FUNCTION_BLOCK ASSEMBLE_AL_FROM_AX (* this Function combines the 64 AX (BOOL) adapters to a AL (LWORD) *)
  (* Standard: 61499-2; Description: Copyright (c) 2026 Meisterschulen am Ostbahnhof SPDX-License-Identifier: EPL-2.0 *)
  (* Version 1.0, 2026-05-16, Franz Höpfinger, Meisterschulen am Ostbahnhof, initial API and implementation and/or initial documentation *)
  PACKAGE adapter::assembling;
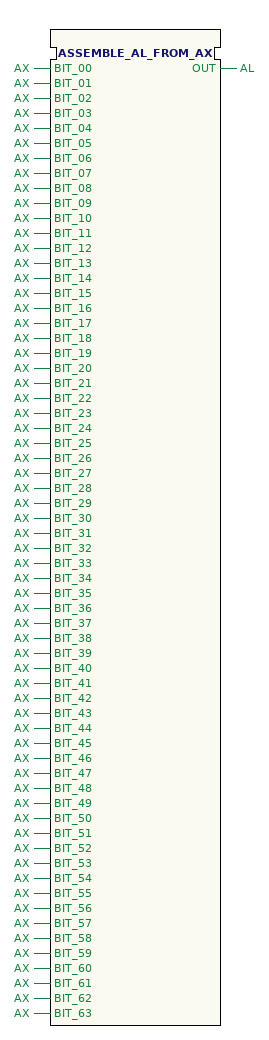
  SOCKETS
    BIT_00 : adapter::types::unidirectional::AX; (* Bool Bit 0 *)
    BIT_01 : adapter::types::unidirectional::AX; (* Bool Bit 1 *)
    BIT_02 : adapter::types::unidirectional::AX; (* Bool Bit 2 *)
    BIT_03 : adapter::types::unidirectional::AX; (* Bool Bit 3 *)
    BIT_04 : adapter::types::unidirectional::AX; (* Bool Bit 4 *)
    BIT_05 : adapter::types::unidirectional::AX; (* Bool Bit 5 *)
    BIT_06 : adapter::types::unidirectional::AX; (* Bool Bit 6 *)
    BIT_07 : adapter::types::unidirectional::AX; (* Bool Bit 7 *)
    BIT_08 : adapter::types::unidirectional::AX; (* Bool Bit 8 *)
    BIT_09 : adapter::types::unidirectional::AX; (* Bool Bit 9 *)
    BIT_10 : adapter::types::unidirectional::AX; (* Bool Bit 10 *)
    BIT_11 : adapter::types::unidirectional::AX; (* Bool Bit 11 *)
    BIT_12 : adapter::types::unidirectional::AX; (* Bool Bit 12 *)
    BIT_13 : adapter::types::unidirectional::AX; (* Bool Bit 13 *)
    BIT_14 : adapter::types::unidirectional::AX; (* Bool Bit 14 *)
    BIT_15 : adapter::types::unidirectional::AX; (* Bool Bit 15 *)
    BIT_16 : adapter::types::unidirectional::AX; (* Bool Bit 16 *)
    BIT_17 : adapter::types::unidirectional::AX; (* Bool Bit 17 *)
    BIT_18 : adapter::types::unidirectional::AX; (* Bool Bit 18 *)
    BIT_19 : adapter::types::unidirectional::AX; (* Bool Bit 19 *)
    BIT_20 : adapter::types::unidirectional::AX; (* Bool Bit 20 *)
    BIT_21 : adapter::types::unidirectional::AX; (* Bool Bit 21 *)
    BIT_22 : adapter::types::unidirectional::AX; (* Bool Bit 22 *)
    BIT_23 : adapter::types::unidirectional::AX; (* Bool Bit 23 *)
    BIT_24 : adapter::types::unidirectional::AX; (* Bool Bit 24 *)
    BIT_25 : adapter::types::unidirectional::AX; (* Bool Bit 25 *)
    BIT_26 : adapter::types::unidirectional::AX; (* Bool Bit 26 *)
    BIT_27 : adapter::types::unidirectional::AX; (* Bool Bit 27 *)
    BIT_28 : adapter::types::unidirectional::AX; (* Bool Bit 28 *)
    BIT_29 : adapter::types::unidirectional::AX; (* Bool Bit 29 *)
    BIT_30 : adapter::types::unidirectional::AX; (* Bool Bit 30 *)
    BIT_31 : adapter::types::unidirectional::AX; (* Bool Bit 31 *)
    BIT_32 : adapter::types::unidirectional::AX; (* Bool Bit 32 *)
    BIT_33 : adapter::types::unidirectional::AX; (* Bool Bit 33 *)
    BIT_34 : adapter::types::unidirectional::AX; (* Bool Bit 34 *)
    BIT_35 : adapter::types::unidirectional::AX; (* Bool Bit 35 *)
    BIT_36 : adapter::types::unidirectional::AX; (* Bool Bit 36 *)
    BIT_37 : adapter::types::unidirectional::AX; (* Bool Bit 37 *)
    BIT_38 : adapter::types::unidirectional::AX; (* Bool Bit 38 *)
    BIT_39 : adapter::types::unidirectional::AX; (* Bool Bit 39 *)
    BIT_40 : adapter::types::unidirectional::AX; (* Bool Bit 40 *)
    BIT_41 : adapter::types::unidirectional::AX; (* Bool Bit 41 *)
    BIT_42 : adapter::types::unidirectional::AX; (* Bool Bit 42 *)
    BIT_43 : adapter::types::unidirectional::AX; (* Bool Bit 43 *)
    BIT_44 : adapter::types::unidirectional::AX; (* Bool Bit 44 *)
    BIT_45 : adapter::types::unidirectional::AX; (* Bool Bit 45 *)
    BIT_46 : adapter::types::unidirectional::AX; (* Bool Bit 46 *)
    BIT_47 : adapter::types::unidirectional::AX; (* Bool Bit 47 *)
    BIT_48 : adapter::types::unidirectional::AX; (* Bool Bit 48 *)
    BIT_49 : adapter::types::unidirectional::AX; (* Bool Bit 49 *)
    BIT_50 : adapter::types::unidirectional::AX; (* Bool Bit 50 *)
    BIT_51 : adapter::types::unidirectional::AX; (* Bool Bit 51 *)
    BIT_52 : adapter::types::unidirectional::AX; (* Bool Bit 52 *)
    BIT_53 : adapter::types::unidirectional::AX; (* Bool Bit 53 *)
    BIT_54 : adapter::types::unidirectional::AX; (* Bool Bit 54 *)
    BIT_55 : adapter::types::unidirectional::AX; (* Bool Bit 55 *)
    BIT_56 : adapter::types::unidirectional::AX; (* Bool Bit 56 *)
    BIT_57 : adapter::types::unidirectional::AX; (* Bool Bit 57 *)
    BIT_58 : adapter::types::unidirectional::AX; (* Bool Bit 58 *)
    BIT_59 : adapter::types::unidirectional::AX; (* Bool Bit 59 *)
    BIT_60 : adapter::types::unidirectional::AX; (* Bool Bit 60 *)
    BIT_61 : adapter::types::unidirectional::AX; (* Bool Bit 61 *)
    BIT_62 : adapter::types::unidirectional::AX; (* Bool Bit 62 *)
    BIT_63 : adapter::types::unidirectional::AX; (* Bool Bit 63 *)
  END_SOCKETS
  PLUGS
    OUT : adapter::types::unidirectional::AL; (* LWORD Output *)
  END_PLUGS
  FBS
    ASSEMBLE_LWORD_FROM_BOOLS : eclipse4diac::utils::assembling::ASSEMBLE_LWORD_FROM_BOOLS;
    E_D_FF_ANY : iec61499::events::E_D_FF_ANY;
  END_FBS
  EVENT_CONNECTIONS
    BIT_00.E1 TO ASSEMBLE_LWORD_FROM_BOOLS.REQ;
    BIT_01.E1 TO ASSEMBLE_LWORD_FROM_BOOLS.REQ;
    BIT_02.E1 TO ASSEMBLE_LWORD_FROM_BOOLS.REQ;
    BIT_03.E1 TO ASSEMBLE_LWORD_FROM_BOOLS.REQ;
    BIT_04.E1 TO ASSEMBLE_LWORD_FROM_BOOLS.REQ;
    BIT_05.E1 TO ASSEMBLE_LWORD_FROM_BOOLS.REQ;
    BIT_06.E1 TO ASSEMBLE_LWORD_FROM_BOOLS.REQ;
    BIT_07.E1 TO ASSEMBLE_LWORD_FROM_BOOLS.REQ;
    BIT_08.E1 TO ASSEMBLE_LWORD_FROM_BOOLS.REQ;
    BIT_09.E1 TO ASSEMBLE_LWORD_FROM_BOOLS.REQ;
    BIT_10.E1 TO ASSEMBLE_LWORD_FROM_BOOLS.REQ;
    BIT_11.E1 TO ASSEMBLE_LWORD_FROM_BOOLS.REQ;
    BIT_12.E1 TO ASSEMBLE_LWORD_FROM_BOOLS.REQ;
    BIT_13.E1 TO ASSEMBLE_LWORD_FROM_BOOLS.REQ;
    BIT_14.E1 TO ASSEMBLE_LWORD_FROM_BOOLS.REQ;
    BIT_15.E1 TO ASSEMBLE_LWORD_FROM_BOOLS.REQ;
    BIT_16.E1 TO ASSEMBLE_LWORD_FROM_BOOLS.REQ;
    BIT_17.E1 TO ASSEMBLE_LWORD_FROM_BOOLS.REQ;
    BIT_18.E1 TO ASSEMBLE_LWORD_FROM_BOOLS.REQ;
    BIT_19.E1 TO ASSEMBLE_LWORD_FROM_BOOLS.REQ;
    BIT_20.E1 TO ASSEMBLE_LWORD_FROM_BOOLS.REQ;
    BIT_21.E1 TO ASSEMBLE_LWORD_FROM_BOOLS.REQ;
    BIT_22.E1 TO ASSEMBLE_LWORD_FROM_BOOLS.REQ;
    BIT_23.E1 TO ASSEMBLE_LWORD_FROM_BOOLS.REQ;
    BIT_24.E1 TO ASSEMBLE_LWORD_FROM_BOOLS.REQ;
    BIT_25.E1 TO ASSEMBLE_LWORD_FROM_BOOLS.REQ;
    BIT_26.E1 TO ASSEMBLE_LWORD_FROM_BOOLS.REQ;
    BIT_27.E1 TO ASSEMBLE_LWORD_FROM_BOOLS.REQ;
    BIT_28.E1 TO ASSEMBLE_LWORD_FROM_BOOLS.REQ;
    BIT_29.E1 TO ASSEMBLE_LWORD_FROM_BOOLS.REQ;
    BIT_30.E1 TO ASSEMBLE_LWORD_FROM_BOOLS.REQ;
    BIT_31.E1 TO ASSEMBLE_LWORD_FROM_BOOLS.REQ;
    BIT_32.E1 TO ASSEMBLE_LWORD_FROM_BOOLS.REQ;
    BIT_33.E1 TO ASSEMBLE_LWORD_FROM_BOOLS.REQ;
    BIT_34.E1 TO ASSEMBLE_LWORD_FROM_BOOLS.REQ;
    BIT_35.E1 TO ASSEMBLE_LWORD_FROM_BOOLS.REQ;
    BIT_36.E1 TO ASSEMBLE_LWORD_FROM_BOOLS.REQ;
    BIT_37.E1 TO ASSEMBLE_LWORD_FROM_BOOLS.REQ;
    BIT_38.E1 TO ASSEMBLE_LWORD_FROM_BOOLS.REQ;
    BIT_39.E1 TO ASSEMBLE_LWORD_FROM_BOOLS.REQ;
    BIT_40.E1 TO ASSEMBLE_LWORD_FROM_BOOLS.REQ;
    BIT_41.E1 TO ASSEMBLE_LWORD_FROM_BOOLS.REQ;
    BIT_42.E1 TO ASSEMBLE_LWORD_FROM_BOOLS.REQ;
    BIT_43.E1 TO ASSEMBLE_LWORD_FROM_BOOLS.REQ;
    BIT_44.E1 TO ASSEMBLE_LWORD_FROM_BOOLS.REQ;
    BIT_45.E1 TO ASSEMBLE_LWORD_FROM_BOOLS.REQ;
    BIT_46.E1 TO ASSEMBLE_LWORD_FROM_BOOLS.REQ;
    BIT_47.E1 TO ASSEMBLE_LWORD_FROM_BOOLS.REQ;
    BIT_48.E1 TO ASSEMBLE_LWORD_FROM_BOOLS.REQ;
    BIT_49.E1 TO ASSEMBLE_LWORD_FROM_BOOLS.REQ;
    BIT_50.E1 TO ASSEMBLE_LWORD_FROM_BOOLS.REQ;
    BIT_51.E1 TO ASSEMBLE_LWORD_FROM_BOOLS.REQ;
    BIT_52.E1 TO ASSEMBLE_LWORD_FROM_BOOLS.REQ;
    BIT_53.E1 TO ASSEMBLE_LWORD_FROM_BOOLS.REQ;
    BIT_54.E1 TO ASSEMBLE_LWORD_FROM_BOOLS.REQ;
    BIT_55.E1 TO ASSEMBLE_LWORD_FROM_BOOLS.REQ;
    BIT_56.E1 TO ASSEMBLE_LWORD_FROM_BOOLS.REQ;
    BIT_57.E1 TO ASSEMBLE_LWORD_FROM_BOOLS.REQ;
    BIT_58.E1 TO ASSEMBLE_LWORD_FROM_BOOLS.REQ;
    BIT_59.E1 TO ASSEMBLE_LWORD_FROM_BOOLS.REQ;
    BIT_60.E1 TO ASSEMBLE_LWORD_FROM_BOOLS.REQ;
    BIT_61.E1 TO ASSEMBLE_LWORD_FROM_BOOLS.REQ;
    BIT_62.E1 TO ASSEMBLE_LWORD_FROM_BOOLS.REQ;
    BIT_63.E1 TO ASSEMBLE_LWORD_FROM_BOOLS.REQ;
    ASSEMBLE_LWORD_FROM_BOOLS.CNF TO E_D_FF_ANY.CLK;
    E_D_FF_ANY.EO TO OUT.E1;
  END_CONNECTIONS
  DATA_CONNECTIONS
    ASSEMBLE_LWORD_FROM_BOOLS. TO E_D_FF_ANY.D;
    E_D_FF_ANY.Q TO OUT.D1;
    BIT_63.D1 TO ASSEMBLE_LWORD_FROM_BOOLS.BIT_63;
    BIT_62.D1 TO ASSEMBLE_LWORD_FROM_BOOLS.BIT_62;
    BIT_61.D1 TO ASSEMBLE_LWORD_FROM_BOOLS.BIT_61;
    BIT_60.D1 TO ASSEMBLE_LWORD_FROM_BOOLS.BIT_60;
    BIT_59.D1 TO ASSEMBLE_LWORD_FROM_BOOLS.BIT_59;
    BIT_58.D1 TO ASSEMBLE_LWORD_FROM_BOOLS.BIT_58;
    BIT_57.D1 TO ASSEMBLE_LWORD_FROM_BOOLS.BIT_57;
    BIT_56.D1 TO ASSEMBLE_LWORD_FROM_BOOLS.BIT_56;
    BIT_55.D1 TO ASSEMBLE_LWORD_FROM_BOOLS.BIT_55;
    BIT_54.D1 TO ASSEMBLE_LWORD_FROM_BOOLS.BIT_54;
    BIT_53.D1 TO ASSEMBLE_LWORD_FROM_BOOLS.BIT_53;
    BIT_52.D1 TO ASSEMBLE_LWORD_FROM_BOOLS.BIT_52;
    BIT_51.D1 TO ASSEMBLE_LWORD_FROM_BOOLS.BIT_51;
    BIT_50.D1 TO ASSEMBLE_LWORD_FROM_BOOLS.BIT_50;
    BIT_49.D1 TO ASSEMBLE_LWORD_FROM_BOOLS.BIT_49;
    BIT_48.D1 TO ASSEMBLE_LWORD_FROM_BOOLS.BIT_48;
    BIT_47.D1 TO ASSEMBLE_LWORD_FROM_BOOLS.BIT_47;
    BIT_46.D1 TO ASSEMBLE_LWORD_FROM_BOOLS.BIT_46;
    BIT_45.D1 TO ASSEMBLE_LWORD_FROM_BOOLS.BIT_45;
    BIT_44.D1 TO ASSEMBLE_LWORD_FROM_BOOLS.BIT_44;
    BIT_43.D1 TO ASSEMBLE_LWORD_FROM_BOOLS.BIT_43;
    BIT_42.D1 TO ASSEMBLE_LWORD_FROM_BOOLS.BIT_42;
    BIT_41.D1 TO ASSEMBLE_LWORD_FROM_BOOLS.BIT_41;
    BIT_40.D1 TO ASSEMBLE_LWORD_FROM_BOOLS.BIT_40;
    BIT_39.D1 TO ASSEMBLE_LWORD_FROM_BOOLS.BIT_39;
    BIT_38.D1 TO ASSEMBLE_LWORD_FROM_BOOLS.BIT_38;
    BIT_37.D1 TO ASSEMBLE_LWORD_FROM_BOOLS.BIT_37;
    BIT_36.D1 TO ASSEMBLE_LWORD_FROM_BOOLS.BIT_36;
    BIT_35.D1 TO ASSEMBLE_LWORD_FROM_BOOLS.BIT_35;
    BIT_34.D1 TO ASSEMBLE_LWORD_FROM_BOOLS.BIT_34;
    BIT_33.D1 TO ASSEMBLE_LWORD_FROM_BOOLS.BIT_33;
    BIT_32.D1 TO ASSEMBLE_LWORD_FROM_BOOLS.BIT_32;
    BIT_31.D1 TO ASSEMBLE_LWORD_FROM_BOOLS.BIT_31;
    BIT_30.D1 TO ASSEMBLE_LWORD_FROM_BOOLS.BIT_30;
    BIT_29.D1 TO ASSEMBLE_LWORD_FROM_BOOLS.BIT_29;
    BIT_28.D1 TO ASSEMBLE_LWORD_FROM_BOOLS.BIT_28;
    BIT_27.D1 TO ASSEMBLE_LWORD_FROM_BOOLS.BIT_27;
    BIT_26.D1 TO ASSEMBLE_LWORD_FROM_BOOLS.BIT_26;
    BIT_25.D1 TO ASSEMBLE_LWORD_FROM_BOOLS.BIT_25;
    BIT_24.D1 TO ASSEMBLE_LWORD_FROM_BOOLS.BIT_24;
    BIT_23.D1 TO ASSEMBLE_LWORD_FROM_BOOLS.BIT_23;
    BIT_22.D1 TO ASSEMBLE_LWORD_FROM_BOOLS.BIT_22;
    BIT_21.D1 TO ASSEMBLE_LWORD_FROM_BOOLS.BIT_21;
    BIT_20.D1 TO ASSEMBLE_LWORD_FROM_BOOLS.BIT_20;
    BIT_19.D1 TO ASSEMBLE_LWORD_FROM_BOOLS.BIT_19;
    BIT_18.D1 TO ASSEMBLE_LWORD_FROM_BOOLS.BIT_18;
    BIT_17.D1 TO ASSEMBLE_LWORD_FROM_BOOLS.BIT_17;
    BIT_16.D1 TO ASSEMBLE_LWORD_FROM_BOOLS.BIT_16;
    BIT_15.D1 TO ASSEMBLE_LWORD_FROM_BOOLS.BIT_15;
    BIT_14.D1 TO ASSEMBLE_LWORD_FROM_BOOLS.BIT_14;
    BIT_13.D1 TO ASSEMBLE_LWORD_FROM_BOOLS.BIT_13;
    BIT_12.D1 TO ASSEMBLE_LWORD_FROM_BOOLS.BIT_12;
    BIT_11.D1 TO ASSEMBLE_LWORD_FROM_BOOLS.BIT_11;
    BIT_10.D1 TO ASSEMBLE_LWORD_FROM_BOOLS.BIT_10;
    BIT_09.D1 TO ASSEMBLE_LWORD_FROM_BOOLS.BIT_09;
    BIT_08.D1 TO ASSEMBLE_LWORD_FROM_BOOLS.BIT_08;
    BIT_07.D1 TO ASSEMBLE_LWORD_FROM_BOOLS.BIT_07;
    BIT_06.D1 TO ASSEMBLE_LWORD_FROM_BOOLS.BIT_06;
    BIT_05.D1 TO ASSEMBLE_LWORD_FROM_BOOLS.BIT_05;
    BIT_04.D1 TO ASSEMBLE_LWORD_FROM_BOOLS.BIT_04;
    BIT_03.D1 TO ASSEMBLE_LWORD_FROM_BOOLS.BIT_03;
    BIT_02.D1 TO ASSEMBLE_LWORD_FROM_BOOLS.BIT_02;
    BIT_01.D1 TO ASSEMBLE_LWORD_FROM_BOOLS.BIT_01;
    BIT_00.D1 TO ASSEMBLE_LWORD_FROM_BOOLS.BIT_00;
  END_CONNECTIONS
END_FUNCTION_BLOCK
